// TIA Portal V21 export
DATA_BLOCK "PhtRecipe"   // DB1218
{ S7_Optimized_Access := 'FALSE' }
// stored: AutoNumber false
   VAR
      HoldPressure : Real := 1.33;
      PressureStabilizeTime : Int := 30;
      AcceptableLeakage : Real := 0.2;
      PressureHoldTime : Int := 1;
      ReleasePressure : Real := 0.1;
   END_VAR
BEGIN
END_DATA_BLOCK
